PROGRAM pouS4Warnings
VAR
	
idbMsgWarn: FB_CheckMessageBounds;
END_VAR

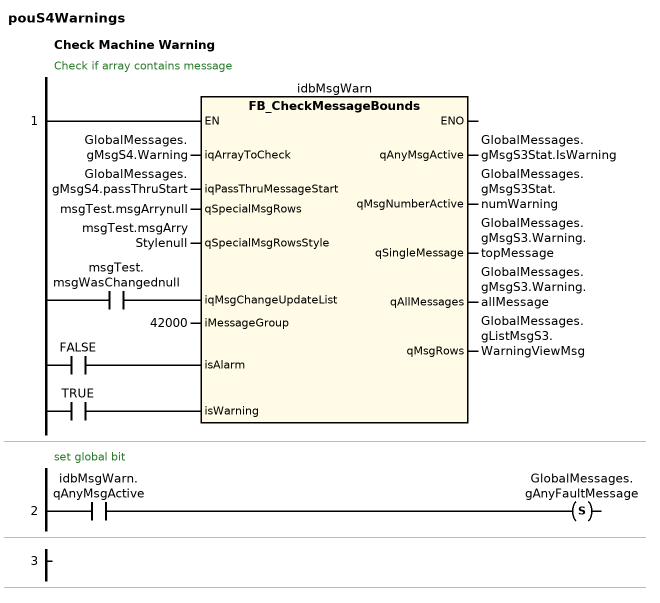
// NETWORK 1: Check Machine Warning
// Check if array contains message
idbMsgWarn(
    iqArrayToCheck := GlobalMessages.gMsgS4.Warning,
    iqPassThruMessageStart := GlobalMessages.gMsgS4.passThruStart,
    qSpecialMsgRows := msgTest.msgArrynull,
    qSpecialMsgRowsStyle := msgTest.msgArryStylenull,
    iqMsgChangeUpdateList := msgTest.msgWasChangednull,
    iMessageGroup := 42000,
    isAlarm := FALSE,
    isWarning := TRUE,
    qAnyMsgActive => GlobalMessages.gMsgS3Stat.IsWarning,
    qMsgNumberActive => GlobalMessages.gMsgS3Stat.numWarning,
    qSingleMessage => GlobalMessages.gMsgS3.Warning.topMessage,
    qAllMessages => GlobalMessages.gMsgS3.Warning.allMessage,
    qMsgRows => GlobalMessages.gListMsgS3.WarningViewMsg); // FB_CheckMessageBounds

// NETWORK 2
// set global bit
GlobalMessages.gAnyFaultMessage S= idbMsgWarn.qAnyMsgActive;

// NETWORK 3

END_PROGRAM

(* stored: Version 1.1.0.1, ProductVersion 3.1.4024.12
   POU pouS4Warnings: Id {9c66757e-dfa8-4e10-bfdf-e4170f7eccb8}, SpecialFunc None *)
